SUBAPPLICATION SlurryTanker (* Subapplication Type *)
  (* Standard: 61499-2 *)
  (* Version 1.0, 2023-02-11, franz *)
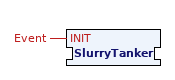
  EVENT_INPUT
    INIT;
  END_EVENT
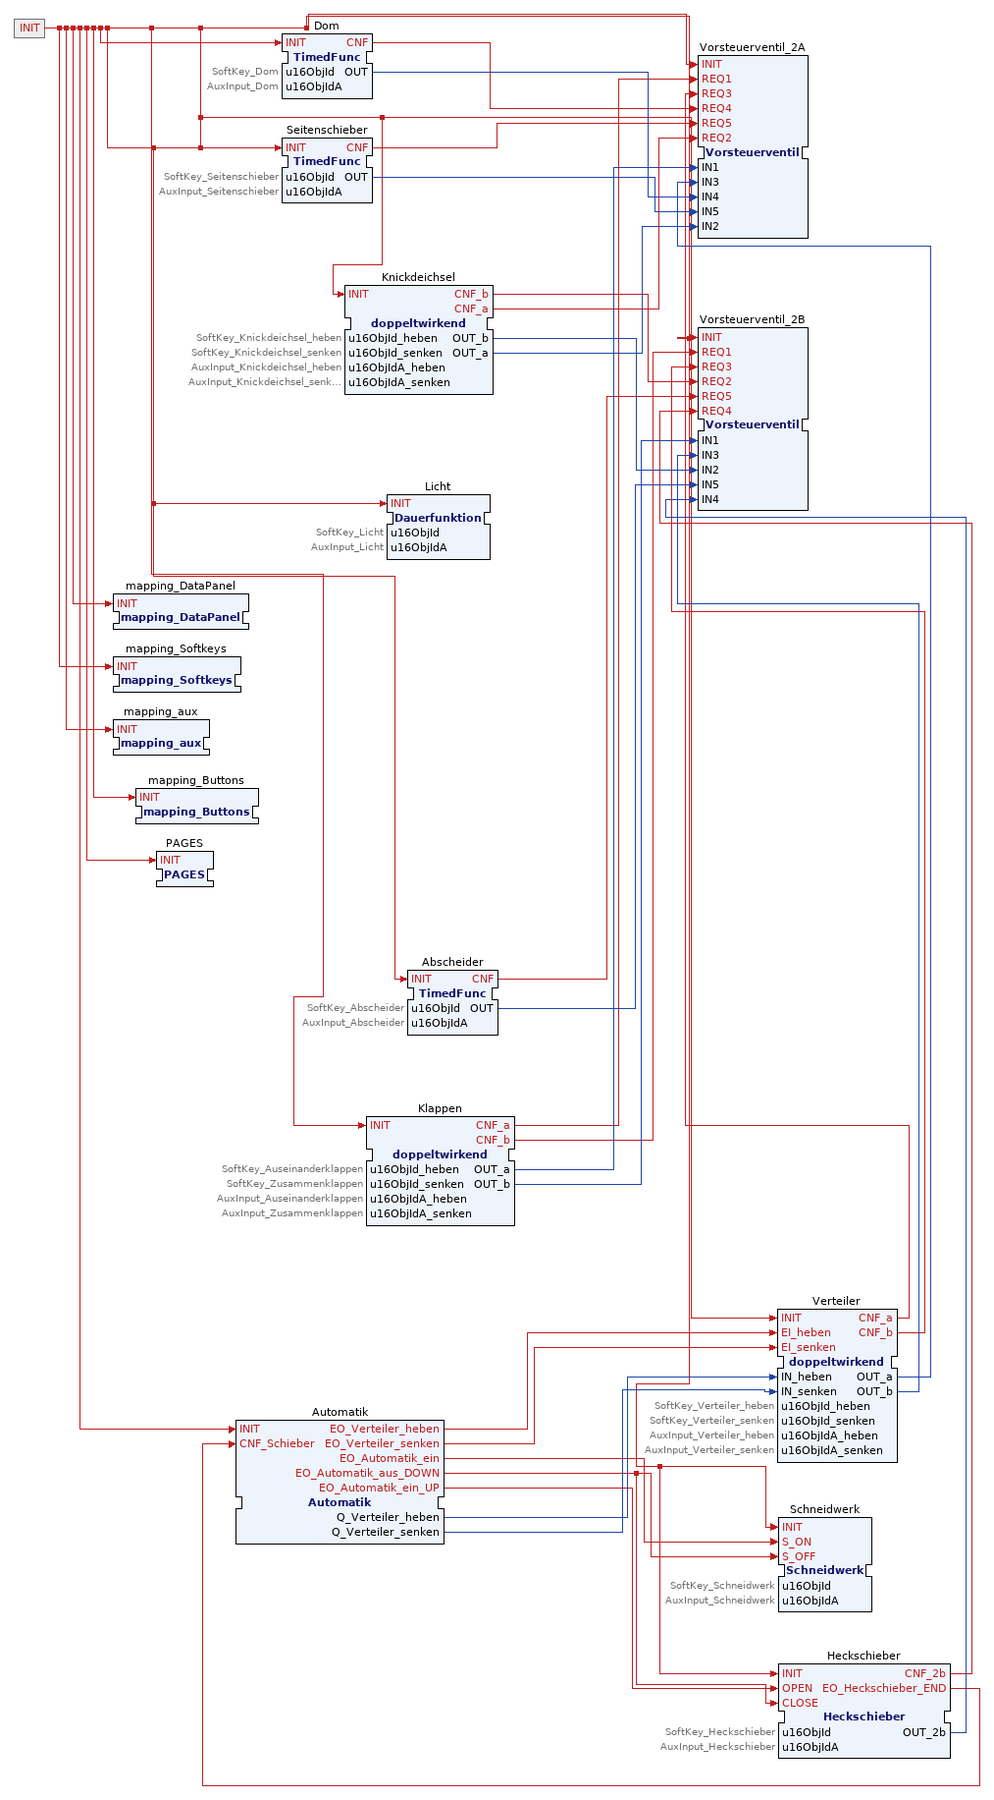
  (* Group func: *)
  (* Group Vorsteuerventile: Vorsteuerventile *)
  (* Group Vorgewendeautomatik: Vorgewendeautomatik *)
  SUBAPPS
    mapping_Softkeys : mapping_Softkeys; {SET_ATTRIBUTE(GroupName, func)}
    mapping_DataPanel : mapping_DataPanel; {SET_ATTRIBUTE(GroupName, func)}
    mapping_aux : mapping_aux; {SET_ATTRIBUTE(GroupName, func)}
    Automatik : Automatik; {SET_ATTRIBUTE(GroupName, Vorgewendeautomatik)}
    PAGES : PAGES; {SET_ATTRIBUTE(GroupName, func)}
    mapping_Buttons : mapping_Buttons; {SET_ATTRIBUTE(GroupName, func)}
    Dom : TimedFunc(u16ObjId := SoftKey_Dom, u16ObjIdA := AuxInput_Dom); {SET_ATTRIBUTE(GroupName, func)}
    Seitenschieber : TimedFunc(u16ObjId := SoftKey_Seitenschieber, u16ObjIdA := AuxInput_Seitenschieber); {SET_ATTRIBUTE(GroupName, func)}
    Klappen : doppeltwirkend(u16ObjId_heben := SoftKey_Auseinanderklappen, u16ObjId_senken := SoftKey_Zusammenklappen, u16ObjIdA_heben := AuxInput_Auseinanderklappen, u16ObjIdA_senken := AuxInput_Zusammenklappen); {SET_ATTRIBUTE(GroupName, func)}
    Verteiler : doppeltwirkend(u16ObjId_heben := SoftKey_Verteiler_heben, u16ObjId_senken := SoftKey_Verteiler_senken, u16ObjIdA_heben := AuxInput_Verteiler_heben, u16ObjIdA_senken := AuxInput_Verteiler_senken); {SET_ATTRIBUTE(GroupName, Vorgewendeautomatik)}
    Vorsteuerventil_2A : Vorsteuerventil; {SET_ATTRIBUTE(GroupName, Vorsteuerventile)}
    Vorsteuerventil_2B : Vorsteuerventil; {SET_ATTRIBUTE(GroupName, Vorsteuerventile)}
    Knickdeichsel : doppeltwirkend(u16ObjId_heben := SoftKey_Knickdeichsel_heben, u16ObjId_senken := SoftKey_Knickdeichsel_senken, u16ObjIdA_heben := AuxInput_Knickdeichsel_heben, u16ObjIdA_senken := AuxInput_Knickdeichsel_senken); {SET_ATTRIBUTE(GroupName, func)}
    Licht : Dauerfunktion(u16ObjId := SoftKey_Licht, u16ObjIdA := AuxInput_Licht); {SET_ATTRIBUTE(GroupName, func)}
    Abscheider : TimedFunc(u16ObjId := SoftKey_Abscheider, u16ObjIdA := AuxInput_Abscheider); {SET_ATTRIBUTE(GroupName, func)}
    Schneidwerk : Schneidwerk(u16ObjId := SoftKey_Schneidwerk, u16ObjIdA := AuxInput_Schneidwerk); {SET_ATTRIBUTE(GroupName, Vorgewendeautomatik)}
    Heckschieber : Heckschieber(u16ObjId := SoftKey_Heckschieber, u16ObjIdA := AuxInput_Heckschieber); {SET_ATTRIBUTE(GroupName, Vorgewendeautomatik)}
  END_SUBAPPS
  EVENT_CONNECTIONS
    INIT TO mapping_Softkeys.INIT;
    INIT TO mapping_aux.INIT;
    INIT TO mapping_DataPanel.INIT;
    INIT TO Automatik.INIT;
    INIT TO PAGES.INIT;
    INIT TO mapping_Buttons.INIT;
    INIT TO Dom.INIT;
    INIT TO Seitenschieber.INIT;
    INIT TO Klappen.INIT;
    INIT TO Verteiler.INIT;
    Automatik.EO_Verteiler_heben TO Verteiler.EI_heben;
    Automatik.EO_Verteiler_senken TO Verteiler.EI_senken;
    INIT TO Vorsteuerventil_2A.INIT;
    Klappen.CNF_a TO Vorsteuerventil_2A.REQ1;
    Verteiler.CNF_a TO Vorsteuerventil_2A.REQ3;
    Dom.CNF TO Vorsteuerventil_2A.REQ4;
    Seitenschieber.CNF TO Vorsteuerventil_2A.REQ5;
    INIT TO Vorsteuerventil_2B.INIT;
    Klappen.CNF_b TO Vorsteuerventil_2B.REQ1;
    Verteiler.CNF_b TO Vorsteuerventil_2B.REQ3;
    INIT TO Knickdeichsel.INIT;
    Knickdeichsel.CNF_b TO Vorsteuerventil_2B.REQ2;
    Knickdeichsel.CNF_a TO Vorsteuerventil_2A.REQ2;
    INIT TO Licht.INIT;
    INIT TO Abscheider.INIT;
    Abscheider.CNF TO Vorsteuerventil_2B.REQ5;
    INIT TO Schneidwerk.INIT;
    Automatik.EO_Automatik_ein TO Schneidwerk.S_ON;
    Automatik.EO_Automatik_aus_DOWN TO Schneidwerk.S_OFF;
    INIT TO Heckschieber.INIT;
    Automatik.EO_Automatik_ein_UP TO Heckschieber.OPEN;
    Automatik.EO_Automatik_aus_DOWN TO Heckschieber.CLOSE;
    Heckschieber.CNF_2b TO Vorsteuerventil_2B.REQ4;
    Heckschieber.EO_Heckschieber_END TO Automatik.CNF_Schieber;
  END_CONNECTIONS
  DATA_CONNECTIONS
    Automatik.Q_Verteiler_heben TO Verteiler.IN_heben;
    Automatik.Q_Verteiler_senken TO Verteiler.IN_senken;
    Klappen.OUT_a TO Vorsteuerventil_2A.IN1;
    Verteiler.OUT_a TO Vorsteuerventil_2A.IN3;
    Dom.OUT TO Vorsteuerventil_2A.IN4;
    Seitenschieber.OUT TO Vorsteuerventil_2A.IN5;
    Klappen.OUT_b TO Vorsteuerventil_2B.IN1;
    Verteiler.OUT_b TO Vorsteuerventil_2B.IN3;
    Knickdeichsel.OUT_b TO Vorsteuerventil_2B.IN2;
    Knickdeichsel.OUT_a TO Vorsteuerventil_2A.IN2;
    Abscheider.OUT TO Vorsteuerventil_2B.IN5;
    Heckschieber.OUT_2b TO Vorsteuerventil_2B.IN4;
  END_CONNECTIONS
END_SUBAPPLICATION
